// Mitsubishi GX Works2 project: test   PLC: FX1S

PROGRAM MAIN
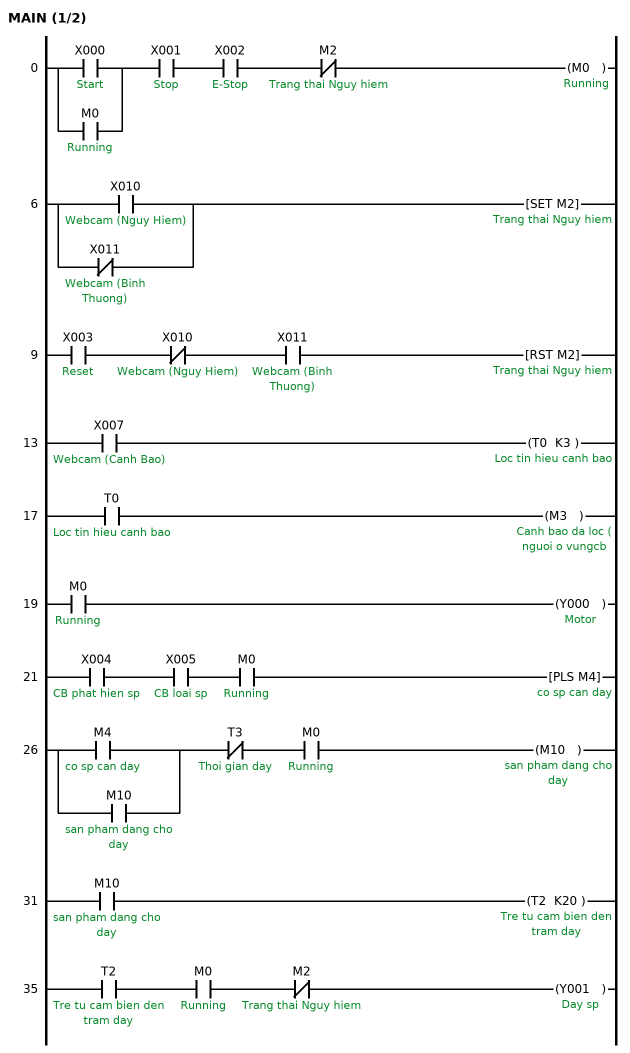
0     LD      X000  ; Start
      OR      M0  ; Running
      AND     X001  ; Stop
      AND     X002  ; E-Stop
      ANI     M2  ; Trang thai Nguy hiem
      OUT     M0  ; Running
6     LD      X010  ; Webcam (Nguy Hiem)
      ORI     X011  ; Webcam (Binh Thuong)
      SET     M2  ; Trang thai Nguy hiem
9     LD      X003  ; Reset
      ANI     X010  ; Webcam (Nguy Hiem)
      AND     X011  ; Webcam (Binh Thuong)
      RST     M2  ; Trang thai Nguy hiem
13    LD      X007  ; Webcam (Canh Bao)
      OUT     T0 K3  ; Loc tin hieu canh bao
17    LD      T0  ; Loc tin hieu canh bao
      OUT     M3  ; Canh bao da loc ( nguoi o vungcb
19    LD      M0  ; Running
      OUT     Y000  ; Motor
21    LD      X004  ; CB phat hien sp
      AND     X005  ; CB loai sp
      AND     M0  ; Running
      PLS     M4  ; co sp can day
26    LD      M4  ; co sp can day
      OR      M10  ; san pham dang cho day
      ANI     T3  ; Thoi gian day
      AND     M0  ; Running
      OUT     M10  ; san pham dang cho day
31    LD      M10  ; san pham dang cho day
      OUT     T2 K20  ; Tre tu cam bien den tram day
35    LD      T2  ; Tre tu cam bien den tram day
      AND     M0  ; Running
      ANI     M2  ; Trang thai Nguy hiem
      OUT     Y001  ; Day sp
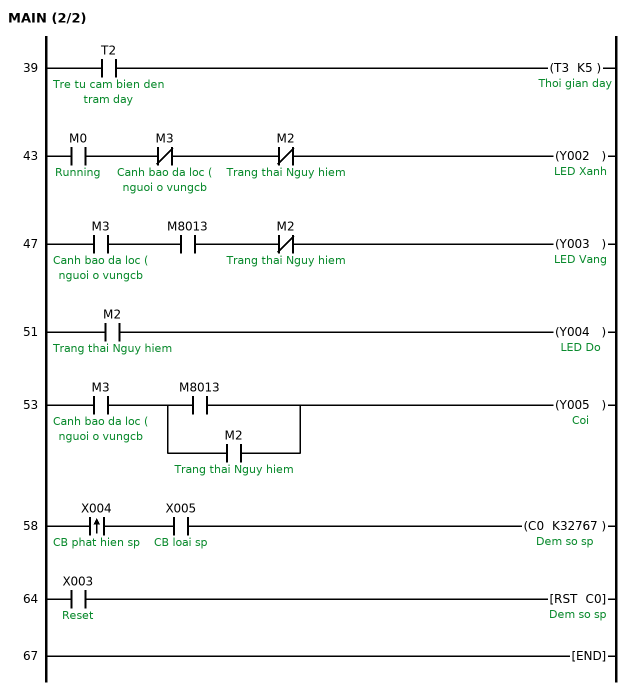
39    LD      T2  ; Tre tu cam bien den tram day
      OUT     T3 K5  ; Thoi gian day
43    LD      M0  ; Running
      ANI     M3  ; Canh bao da loc ( nguoi o vungcb
      ANI     M2  ; Trang thai Nguy hiem
      OUT     Y002  ; LED Xanh
47    LD      M3  ; Canh bao da loc ( nguoi o vungcb
      AND     M8013
      ANI     M2  ; Trang thai Nguy hiem
      OUT     Y003  ; LED Vang
51    LD      M2  ; Trang thai Nguy hiem
      OUT     Y004  ; LED Do
53    LD      M3  ; Canh bao da loc ( nguoi o vungcb
      LD      M8013
      OR      M2  ; Trang thai Nguy hiem
      ANB
      OUT     Y005  ; Coi
58    LDP     X004  ; CB phat hien sp
      AND     X005  ; CB loai sp
      OUT     C0 K32767  ; Dem so sp
64    LD      X003  ; Reset
      RST     C0  ; Dem so sp
67    END
END_PROGRAM

// device comments not shown above
X006  ; Backup
